{attribute addProperty BoxType "EK1100-0000-0018"}
{attribute addProperty Id "Beckhoff_EJ9xxxEK1122Beckhoff_EJ9xxxEK1122_DB893B98162A_0001_EJ9001_0000_0016EJ9001_179A0949162A_0002_EJ9505_0000_0016EJ9505_13AAEB7E344.25A_0003_EJ9576_0000_0018EJ9576_30D5723B21026.25A_0004_EJ9576_0000_0019EJ9576_8602C5C421827.25A_0005_EJ9576_0000_0020EJ9576_EB67CEB421026.25A_0006_EJ9576_0000_0022EJ9576_EEF1625221827.25"}
{attribute addProperty CRC "1712008333"}
{attribute addProperty SizeInBites "922"}
{attribute addProperty SizeInBytes "115.25"}
TYPE Beckhoff_EJ9xxx_660B2C8D EXTENDS EK1100_179A0949 :
STRUCT
	{attribute addProperty Name "Beckhoff_EJ9xxxEK1122"}
	Beckhoff_EJ9xxxEK1122 : Beckhoff_EJ9xxxEK1122_DB893B98;
	{attribute addProperty Name "A_0001_EJ9001_0000_0016"}
	A_0001_EJ9001_0000_0016 : EJ9001_179A0949;
	{attribute addProperty Name "A_0002_EJ9505_0000_0016"}
	A_0002_EJ9505_0000_0016 : EJ9505_13AAEB7E;
	{attribute addProperty Name "A_0003_EJ9576_0000_0018"}
	A_0003_EJ9576_0000_0018 : EJ9576_30D5723B;
	{attribute addProperty Name "A_0004_EJ9576_0000_0019"}
	A_0004_EJ9576_0000_0019 : EJ9576_8602C5C4;
	{attribute addProperty Name "A_0005_EJ9576_0000_0020"}
	A_0005_EJ9576_0000_0020 : EJ9576_EB67CEB4;
	{attribute addProperty Name "A_0006_EJ9576_0000_0022"}
	A_0006_EJ9576_0000_0022 : EJ9576_EEF16252;
END_STRUCT
END_TYPE

(* stored: Version 1.2.0.0, ProductVersion 3.1.4024.9
   DUT Beckhoff_EJ9xxx_660B2C8D: Id {41cf1c5d-6174-4cdb-9abc-633016771691} *)
